{attribute 'qualified_only'}
VAR_GLOBAL
END_VAR

(* stored: Version 1.1.0.1, ProductVersion 3.1.4024.12
   GVL G_OPC: Id {e1bfbbdc-c253-4ef4-aa4a-2d002f8e2c27} *)
